// TIA Portal V16 export
// export: Created 2022-03-28T07:44:08.9013015Z, ExportSetting WithDefaults, DisplayName Totally Integrated Automation Portal, DisplayVersion V16 Update 5, DisplayName TIA Portal Version Control Interface, DisplayVersion V16 Update 2, DisplayName TIA Portal Openness, DisplayVersion V16 Update 5, DisplayName STEP 7 Professional, DisplayVersion V16 Update 5, DisplayName STEP 7 Safety, DisplayVersion V16, DisplayName WinCC Professional, DisplayVersion V16 Update 5
TYPE "udtProgram"
// stored: IsFailsafeCompliant false
   STRUCT
      strName : String[12];
      udtStep { S7_SetPoint := 'True'} : Array[1..10] of "udtStep";
      udtCounter { S7_SetPoint := 'True'} : "udtCounters";
   END_STRUCT;
END_TYPE
